// TIA Portal V19 export
// export: Created 2026-08-09T02:36:23.1467409Z, ExportSetting WithDefaults, DisplayName Totally Integrated Automation Portal, DisplayVersion V19, DisplayName TIA Portal Openness, DisplayVersion V19, DisplayName TIA Portal Version Control Interface, DisplayVersion V19, DisplayName STEP 7 Professional, DisplayVersion V19, DisplayName STEP 7 Safety, DisplayVersion V19, DisplayName WinCC Basic/Comfort/Advanced, DisplayVersion V19, DisplayName WinCC Unified, DisplayVersion V19
FUNCTION_BLOCK "ceD2"   // FB2, LAD
{ S7_Optimized_Access := 'TRUE' }
VERSION : 0.1
// stored: AutoNumber true, IsIECCheckEnabled false, IsRetainMemResEnabled false, MemoryReserve 100, SetENOAutomatically false, UDAEnableTagReadback false
   VAR_INPUT
      in1 : Bool;
      in2 : Bool;
      in3 : Bool;
   END_VAR
   VAR_OUTPUT
      out1 : Bool;
      out2 : Bool;
      out3 : Bool;
   END_VAR
BEGIN

REGION Network 1
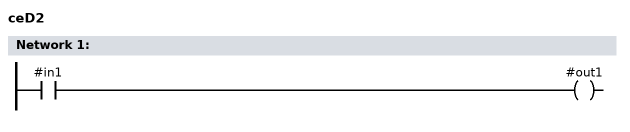
   RUNG wire#powerrail
      Contact( #in1 )
      Coil( #out1 )
   END_RUNG
   // the same network as SCL:
   #out1 := #in1;
END_REGION

NETWORK
TITLE = 

      CALL  R_TRIG, "R_TRIG_DB"
      ( CLK := #in2,
        Q   := #out2
      );




END_FUNCTION_BLOCK
